PROGRAM P_Gang_4_208
VAR
(*Gangen består af to lysgrupper - L2G6 og L1G15
Begge grupper afhænger af samme PIR-input - pir-adr. 6, 7, 8, 9 og 10 - på DALI-linje 2.
Derfor oprettes to adskilte reguleringer med samme PV. Dvs., at knapfunktion og pirfunktion forbliver den samme.

En anden del af af hele gangen styres fra AH4_3. De to dele nabostyres med PIR-signaler over modbus-kommunikation*)
/////////////////////////////////
(*Gangen består af to lysgrupper - 4 og 4 - på to forskellige DALI-linjer - 2 og 1 henh..
Begge grupper afhænger af samme PIR-input - pir-adr. 6, 7, 8, 9 og 10 - på DALI-linje 2.
Derfor oprettes to adskilte reguleringer med samme PV. Dvs., at knapfunktion og pirfunktion forbliver den samme.

En anden del af af hele gangen styres fra AH4_3. De to dele nabostyres med PIR-signaler over modbus-kommunikation*)

	arrfbLysGruppe			: ARRAY [1..2] OF FB_Light_Type_B;
	arrstDaliSetupGruppe	: ARRAY[1..2] OF SH_Light.ST_DALI_RoomSetup := 
	
													[(	byShrtAdr_Prim := 25, 
														byGrpAdr_Prim := 5, 
														eMod_Prim := E_DALIAddressType.Group, 
														byShrtAdr_Sec := 1, 
														byGrpAdr_Sec := 1, 
														eMod_Sec := E_DALIAddressType.Short, 
														//byShrtAdr_Supl := 1,
														//eMod_Supl := E_DALIADDRESSTYPE.Group,
                                                        byGrpAdr_Supl := 1, 
														DALI_LINE_NUM_PRIM := arrDALI_LINE_NUM_LIGHT[1], 
														DALI_LINE_NUM_SEC := 0, //0 = ingen zonestyring/vinduerække
														DALI_LINE_NUM_SUPL := arrDALI_LINE_NUM_PENDANTS[1]),
														
													(	byShrtAdr_Prim := 20, 
														byGrpAdr_Prim := 5, 
														eMod_Prim := E_DALIAddressType.Group, 
														byShrtAdr_Sec := 1, 
														byGrpAdr_Sec := 1, 
														eMod_Sec := E_DALIAddressType.Short, 
														byShrtAdr_Supl := 1, 
														DALI_LINE_NUM_PRIM := arrDALI_LINE_NUM_LIGHT[2], 
														DALI_LINE_NUM_SEC := 0, 
														DALI_LINE_NUM_SUPL := arrDALI_LINE_NUM_PENDANTS[2])];
														
	arrstLiveDataGruppe		: ARRAY [1..2] OF SH_Light.ST_LiveData;
	//stLiveData AT %MB22	: SH_Light.ST_LiveData;
	
	arrRunTuningGruppe: ARRAY[1..2] OF BOOL;
	
	
	
	bTopButtonZone1			: BOOL;
	bTopButtonZone1_Visu	: BOOL;
	bBottomButtonZone1		: BOOL;
	bBottomButtonZone1_Visu	: BOOL;
	bButtonZone2			: BOOL;
	bNeighborRoomsPir		: BOOL;
	fLuxOn					: REAL; 
	fLuxDim					: REAL;
	tPIRDim					: TIME;
	tPIROff					: TIME;
	fOffsetSec				: REAL := 20;

//Digital In
//    bDigitalPir AT %I*      : BOOL ;    

// Sensor Settings
	//fbSensor					: SH_Light.FB_NIKO_P46xx_1Pcs;
	fbSensor					: SH_Light.FB_NIKO_P46xx_3Pcs;
	//bySensorAddr				: BYTE := 17;
	arrSensorAddr				: ARRAY[1..3] OF BYTE := [2,3,4];
	bInitialize					: BOOL := TRUE;
	stDaliSensorSetup			: ST_DALI_NIKOP46SetupData;
	//bInitErr					: BOOL;
	//bInitDone					: BOOL;
	arrInitErr					: ARRAY [1..3] OF BOOL;
	arrInitDone					: ARRAY [1..3] OF BOOL;
	arrSensorScales				: ARRAY [1..10] OF SH_Light.ST_DALI_SensorScaleMode := [	(fMeassureMaxSensor := rMeassure_Zone8, fReadMaxSensor := rRead_Zone8),
																							(fMeassureMaxSensor := rMeassure_Zone8, fReadMaxSensor := rRead_Zone8),	
                                                                                            (fMeassureMaxSensor := rMeassure_Zone8, fReadMaxSensor := rRead_Zone8),																				
																						7(())];
	bCancelHoldTimerOccupancy	: BOOL;
(*	eEventPriorityOccupancy		: E_DALIEventPriority := E_DALIEVENTPRIORITY.Middle;
	nHoldTimerOccupancy			: WORD := 5; // Value in s. 	
	nReportTimerOccupancy		: BYTE := 120; // Value in s, Preset manufacturer value
	nDeadtimeTimerOccupancy		: WORD := 100; // Value in ms, Predefined Value of DALI Standard
	bCancelHoldTimerOccupancy	: BOOL;
	nSensitivityOccupancy		: BYTE:= 3; //setting Sensivity (0..4) 0 (Off), 1 (Min), 2(Low), 3(High) and 4 (Max)

	bEnableLuxEvent				: BOOL;
	eEventPriorityBrightness	: E_DALIEventPriority := E_DALIEVENTPRIORITY.Middle;
	nDeadtimeTimerBrightness	: WORD := 1500; // Value in ms, Predefined Value of DALI Standard
	nHysteresisBrightness		: BYTE := 2; // Value in %
	nHysteresisMinBrightness	: BYTE := 10; // Absolute Value, depending on the manufacturer specific resolution
	nReportTimerBrightness		: BYTE := 120; // Value in s, Preset manufacturer value
*)


//ModbusComm setup
	
	fbWriteSPLuxLevel			: SH_Light.FB_TwoVal_SelectOne_RTrigChange;
	fbWritePirDelayTIme			: SH_Light.FB_TwoVal_SelectOne_RTrigChange;
	stRoomDataPLC				: SH_Light.ST_RoomDataPLC	:=	(	uiPirOffDelayTime	:= 30,
																	uiSpLuxLevel		:= 500,
																	uiPirDimDelayTime	:= 15,
																	uiSpDimLuxLevel		:= 200
																);
	fbBallastOnHours			: SH_Light.FB_CountOnHours;
	bEnableHourCount			: BOOL := TRUE;
	
	//Non-persistent modbus data
	bPirActive_MB			AT%MX60.0	: BOOL;				//bPirLys i gammel kode
	uiActLuxLevel_MB		AT%MB64	: UINT;				//intHMIAktueltLux i gammel kode
	uiActLightLevelPct_MB	AT%MB68	: UINT;				//intDALI_Gruppe1_Lysniveau i gammel kode
	
	//For Conversion
	uiPirOffMinutes						: UINT;
	udTimeScaling						: UDINT := 60000;
	uiLuxOn								: UINT;
	
	//max values checks
	uiMaxLuxLevel						: UINT := 1023;
	uiMaxPirOffMinutes					: UINT := 180;
	
END_VAR

VAR CONSTANT
	Sensor_DALI_LINE_NUM: BYTE := 3;
	arrDALI_LINE_NUM_LIGHT: ARRAY[1..2] OF BYTE := [2,1]; //korrekt rækkefølge nødvendig //rækkefølge og linje 
	arrDALI_LINE_NUM_PENDANTS: ARRAY[1..2] OF BYTE := [0,0]; //korrekt rækkefølge nødvendig. 0 = ingen pendler
END_VAR
VAR PERSISTENT
	stPirSensorData: SH_Light.ST_DALI_Sensor;
	arrstTuneDataGruppe: ARRAY [1..2] OF SH_Light.ST_TuneData_EX;

	uiPirOffDelayTime_MB	AT%MB62	    : UINT;				//intHMI_Pir_SetValue i gammel kode
	uiSPLuxLevel_MB		    AT%MB66     : UINT;				//intHMI_Lux_SetValue i gammel kode
	uiBallastOnHours_MB	    AT%MB70	    : UINT;				//dintHMILysbraendtimer1 i gammel kode
	byOnHoursOverflowCount			    : BYTE;
END_VAR

///////)

A_Buttons();
A_LightCtrl();
A_ModbusComm();
A_Sensor();

ACTION A_Buttons:
bTopButtonZone1		:= bTopButtonZone1_Visu;
bBottomButtonZone1	:= bBottomButtonZone1_Visu;
END_ACTION

ACTION A_LightCtrl:
bNeighborRoomsPir	:=    GVL_AHDataModbus.arrAH_NeighborRoomsPir  [4] [0] OR //2-1 
GVL_AHDataModbus.arrAH_NeighborRoomsPir  [4] [1] OR  //2-1 
GVL_AHDataModbus.arrAH_NeighborRoomsPir  [4] [2] OR //2-1 
GVL_AHDataModbus.arrAH_NeighborRoomsPir  [18] [0] OR//5-1
GVL_AHDataModbus.arrAH_NeighborRoomsPir  [18] [1]OR //5-1
GVL_AHDataModbus.arrAH_NeighborRoomsPir  [5] [0] OR //2-2
GVL_AHDataModbus.arrAH_NeighborRoomsPir  [5] [1] OR //2-2
GVL_AHDataModbus.arrAH_NeighborRoomsPir  [5] [2] OR //2-2
GVL_AHDataModbus.arrAH_NeighborRoomsPir  [5] [3] OR //2-2
GVL_AHDataModbus.arrAH_NeighborRoomsPir  [5] [4] OR //2-2
GVL_AHDataModbus.arrAH_NeighborRoomsPir  [5] [5] OR //2-2
GVL_AHDataModbus.arrAH_NeighborRoomsPir  [9] [0] OR //3-2 
GVL_AHDataModbus.arrAH_NeighborRoomsPir  [9] [1] OR //3-2 
GVL_AHDataModbus.arrAH_NeighborRoomsPir  [9] [2]  OR //3-2 
GVL_AHDataModbus.arrAH_NeighborRoomsPir  [14] [0] OR //4-2 
GVL_AHDataModbus.arrAH_NeighborRoomsPir [14] [1] OR //4-2 
GVL_AHDataModbus.arrAH_NeighborRoomsPir  [19] [0] OR //5-2 
GVL_AHDataModbus.arrAH_NeighborRoomsPir [19] [1] OR //5-2 
GVL_AHDataModbus.arrAH_NeighborRoomsPir [19] [2];  //5-2

                       ;
//gruppe 6
arrfbLysGruppe[1]( 
	nZoneID:= 1, 
	bButtonZone1:= bTopButtonZone1,
	bBottomButtonZone1 := bBottomButtonZone1,
	bTopButtonOverride := (GVL_EnOcean.strEnOceanSwitch_AtriumNiveau_PladeB.bT2_ON OR GVL_EnOcean.strEnOceanSwitch_AtriumNiveau_Service.bT2_ON),
	bBottomButtonOverride := (GVL_EnOcean.strEnOceanSwitch_AtriumNiveau_PladeB.bT2_OFF OR GVL_EnOcean.strEnOceanSwitch_AtriumNiveau_Service.bT2_OFF),
	bButtonZone2:= bButtonZone2,
	bNoButtons := TRUE,
	bNeighborRoomsPir	:=	bNeighborRoomsPir,
	fLuxOn:= fLuxOn, 
	fLuxDim:= fLuxDim, 
	tPIRDim:= tPIRDim, 
	tPIROff:= tPIROff, 
	fOffsetSec:= fOffsetSec, 
	bReInit:= , 
	stDaliSetup:= arrstDaliSetupGruppe[1], 
	ipCommunication_Prim:= P_DALI_Background.arrfbKL6821Communication[arrDALI_LINE_NUM_LIGHT[1]], 
	ipCommunication_Sec:= P_DALI_Background.arrfbKL6821Communication[arrDALI_LINE_NUM_LIGHT[1]], //samme som lyslinjen, hvis den ikke eksisterer
	ipCommunication_Supl:= P_DALI_Background.arrfbKL6821Communication[arrDALI_LINE_NUM_LIGHT[1]],//samme som lyslinjen, hvis den ikke eksisterer 
	fMinOutputPowerLevelRoom:= 15, 
	fMaxOutputPowerLevelRoom:= 100, 
	nCycleTimeInMS:= SH_Light.DALI_Param.nPlcTaskCycleTimeInMS*nDimCmdCycleTimeFactor,  //Used only for dim. Factor=2 makes dimming smooth
	bRunTuning:= arrRunTuningGruppe[1], 
	bOccupiedRoom=> , 
	bError_Prim=> , 
	nError_Prim=> , 
	stTuneData:=arrstTuneDataGruppe[1] , 
	stPirSensorData:= stPirSensorData, 					//samme sensordata
	stLiveData:= arrstLiveDataGruppe[1]);

//gruppe 15	
arrfbLysGruppe[2]( 
	nZoneID:= 1, 
	bButtonZone1:= bTopButtonZone1,
	bBottomButtonZone1 := bBottomButtonZone1,
	bTopButtonOverride := (GVL_EnOcean.strEnOceanSwitch_AtriumNiveau_PladeB.bT2_ON OR GVL_EnOcean.strEnOceanSwitch_AtriumNiveau_Service.bT2_ON),
	bBottomButtonOverride := (GVL_EnOcean.strEnOceanSwitch_AtriumNiveau_PladeB.bT2_OFF OR GVL_EnOcean.strEnOceanSwitch_AtriumNiveau_Service.bT2_OFF),
	bButtonZone2:= bButtonZone2,
	bNoButtons := TRUE,
	bNeighborRoomsPir	:=	bNeighborRoomsPir,
	fLuxOn:= fLuxOn, 
	fLuxDim:= fLuxDim, 
	tPIRDim:= tPIRDim, 
	tPIROff:= tPIROff, 
	fOffsetSec:= fOffsetSec, 
	bReInit:= , 
	stDaliSetup:= arrstDaliSetupGruppe[2], 
	ipCommunication_Prim:= P_DALI_Background.arrfbKL6821Communication[arrDALI_LINE_NUM_LIGHT[2]], 
	ipCommunication_Sec:= P_DALI_Background.arrfbKL6821Communication[arrDALI_LINE_NUM_LIGHT[2]], //samme som lyslinjen, hvis den ikke eksisterer
	ipCommunication_Supl:= P_DALI_Background.arrfbKL6821Communication[arrDALI_LINE_NUM_LIGHT[2]], //samme som lyslinjen, hvis den ikke eksisterer 
	fMinOutputPowerLevelRoom:= 15, 
	fMaxOutputPowerLevelRoom:= 100, 
	nCycleTimeInMS:= SH_Light.DALI_Param.nPlcTaskCycleTimeInMS*nDimCmdCycleTimeFactor,  //Used only for dim. Factor=2 makes dimming smooth
	bRunTuning:= arrRunTuningGruppe[2], 
	bOccupiedRoom=> , 
	bError_Prim=> , 
	nError_Prim=> , 
	stTuneData:=arrstTuneDataGruppe[2] , 
	stPirSensorData:= stPirSensorData, 					//samme sensordata
	stLiveData:= arrstLiveDataGruppe[2]);
END_ACTION

ACTION A_ModbusComm:
//Manage data for modbus communication

//Manage data for read-only in PLC
stRoomDataPLC.bPirActive			:= stPirSensorData.bPrc;
stRoomDataPLC.uiActLuxLevel			:= TO_UINT(TRUNC(stPirSensorData.fBrightness));
stRoomDataPLC.uiActLightLevelPct	:= TO_UINT(TRUNC(arrfbLysGruppe[1].fbBallast.fActlLgtLvl_Prim));
		//stRoomDataPLC.uiActLightLevelPct	:= TO_UINT(TRUNC(fbLys.fbBallast.fActlLgtLvl_Prim)); //if only one group light control
stRoomDataPLC.uiBallastOnHours		:= uiBallastOnHours_MB; //The calculation for BallastOnHours is stored directly to the MB register below


//Assign data for read-only to MB registers
bPirActive_MB		:= stRoomDataPLC.bPirActive;
uiActLuxLevel_MB	:= stRoomDataPLC.uiActLuxLevel;

	//calculate BallastOnHours
	fbBallastOnHours(
		bEnableHourCount	:= bEnableHourCount,
		bPauseCount			:= arrfbLysGruppe[1].fbLightCtrl.bOffZone1,
		uiOnHours			:= uiBallastOnHours_MB,			//OnHours is updated here
		byOverflowCount		:= byOnHoursOverflowCount);


//Manage data for read/write for both PLC and MB registers
fbWriteSPLuxLevel(	nMaxValOut	:= uiMaxLuxLevel,
					nValIn1		:= uiSPLuxLevel_MB,		//nValIn1 takes priotity in case of download or restart
					nValIn2		:= stRoomDataPLC.uiSpLuxLevel,
					nValOut		=> uiLuxOn
				);


fbWritePirDelayTIme(	nMaxValOut	:= uiMaxPirOffMinutes,
						nValIn1		:= uiPirOffDelayTime_MB,		//nValIn1 takes priotity in case of download or restart
						nValIn2		:= stRoomDataPLC.uiPirOffDelayTime,
						nValOut		=> uiPirOffMinutes
					);
					

//Convert read/write modbus data to appropriate datatypes in PLC
fLuxOn	:= TO_REAL(uiLuxOn);			
tPIROff	:= TO_TIME(uiPirOffMinutes*udTimeScaling); //Time conversion defaults to ms

fLuxDim	:= TO_REAL(stRoomDataPLC.uiSpDimLuxLevel);			
tPIRDim	:= TO_TIME(stRoomDataPLC.uiPirDimDelayTime*udTimeScaling); //Time conversion defaults to ms
END_ACTION

ACTION A_Sensor:

fbSensor.ipCommunication := P_DALI_Background.arrfbKL6821Communication[Sensor_DALI_LINE_NUM];

(*//only 1 sensor
fbSensor(
	byShrtAdr:= bySensorAddr,
	bInitialize:= bInitialize, 
	DALI_LINE_NUM:= Sensor_DALI_LINE_NUM, 
 	//bCancelHoldTimerOccupancy:= bCancelHoldTimerOccupancy, 
	stSensorSetup := stDaliSensorSetup,
	bInitErr=> bInitErr, 
	bInitDone=> bInitDone,
	stPirSensorData:= stPirSensorData, 
	arrSensorScales:= arrSensorScales);
	*)

//several sensors	
fbSensor(
	arrShrtAdr:= arrSensorAddr,
	bInitialize:= bInitialize, 
	DALI_LINE_NUM:= Sensor_DALI_LINE_NUM, 
 	//bCancelHoldTimerOccupancy:= bCancelHoldTimerOccupancy, 
	stSensorSetup := stDaliSensorSetup,
	arrInitErr=> arrInitErr, 
	arrInitDone=> arrInitDone,
	stPirSensorData:= stPirSensorData, 
	arrSensorScales:= arrSensorScales);
END_ACTION

END_PROGRAM

(* stored: Version 1.1.0.1
   POU P_Gang_4_208: Id {ba44d9a3-1b28-408f-b76c-8f64851151e8}, SpecialFunc None
   Action A_Buttons: Id {c8d87400-0b27-443d-a1cc-cd273da605bc}
   Action A_LightCtrl: Id {8019beaf-b0b8-4c93-b975-caa6dc202667}
   Action A_ModbusComm: Id {236a9e96-6a69-4fe6-93b4-c524294d51c0}
   Action A_Sensor: Id {fbced804-1b45-4c0b-b2d5-653b53bc209b} *)
